FUNCTION_BLOCK FB_Machine EXTENDS FB_PackML_BaseModule // IMPLEMENTS I_ControlsProductionRate
VAR
    // Sub Modules
    GantryXYZ   : FB_GantryXYZ  := (Name := 'Gantry', LogStateChanges := TRUE);

    //Initial List of Components
    ipComponents_Init : ARRAY[1..Parameters_PackML_Base.MAX_NO_OF_COMPONENTS] OF I_ComponentBase := [];

	//Alarms for this module
	MachineAlarms : ARRAY[1..MACHINE_ALARM_COUNT] OF FB_TcAlarm;

END_VAR

VAR CONSTANT
    MACHINE_ALARM_COUNT : INT := 6;
END_VAR


METHOD PROTECTED Clearing
VAR
	i				: UDINT;
	SubModulesReady : BOOL := TRUE;
END_VAR
CASE SequenceState OF
    0:
        NoStateTasksToComplete := FALSE;
        SequenceState          := SequenceState + 10;
    10:
		//Leave Aborted thanks to this
		MachineAlarms[E_Seedra.EmergencyStop].Clear(0, 0);
        SequenceState := SequenceState + 10;
    20:

		SequenceState := SequenceState + 10;
	30: 
	
		SequenceState := SequenceState + 10;
	40:
		StateTasksComplete := TRUE; 
			 
END_CASE

SUPER^.Clearing();
END_METHOD

METHOD PROTECTED CreateEvents
VAR_INPUT
END_VAR
// Add your event creation here
F_CreateAllEventsInClass(Alarms     := MachineAlarms,
                         ClassSize  := SIZEOF(TC_Events.Seedra),
                         pInitEvent := ADR(TC_EVENTS.Seedra.InitReferenceEvent),
                         Prefix     := Name);
// Super call to base
SUPER^.CreateEvents();
END_METHOD

METHOD CyclicLogic
VAR_INPUT
END_VAR

IF NOT _InitComplete THEN
    _InitComplete := Initialize();
    RETURN;
END_IF

SUPER^.CyclicLogic();

//Here the alarms will raise and clear on its own if the input changes

//NOT GVL_Safety.eStopButton -> We Decouple physical button to Activate
  
IF GVL_Safety.eStopHMI OR NOT GVL_Safety.eStopButton AND NOT MachineAlarms[E_Seedra.EmergencyStop].bRaised THEN
	THIS^.ChangeState(E_PMLCommand.ePMLCommand_Abort);
	RaiseAlarmWithStrings(MachineAlarms[E_Seedra.EmergencyStop],'','');
//	ELSIF NOT GVL_Safety.eStop THEN
//	MachineAlarms[E_Seedra.EmergencyStop].Clear(0, 0);

END_IF
END_METHOD

METHOD PROTECTED Execute
CASE _CurrentMode OF

	//=================================PRODUCTION MODE==================================
	E_PMLUnitMode.ePMLUnitMode_Production:
		CASE SequenceState OF
			0:
				NoStateTasksToComplete := FALSE;

				//Advance Gantry to Resetting (Homing)
				GantryXYZ.ChangeState(E_PMLCommand.ePMLCommand_Start);
				
				SequenceState := SequenceState + 10;
					
			10:
				StateTasksComplete := TRUE;
				StateComplete();
				
			
		END_CASE

	//=================================MAINTENANCE & MANUAL MODE==================================
	E_PMLUnitMode.ePMLUnitMode_Maintenance, E_PMLUnitMode.ePMLUnitMode_Manual:
		;
END_CASE
END_METHOD

//! @summary Provides interlocks for HMI control and updates HMI status information for this module
METHOD PROTECTED HMICommunication

//! @description This method is called cyclically by <c>CyclicLogic()</c>

IF GVL_Safety.eStopHMI THEN
	PackMLBaseModule_HMI.Status.Error := TRUE;
	THIS^._Error := TRUE;
END_IF



SUPER^.HMICommunication();
END_METHOD

METHOD PROTECTED HMIPermissions
//General Mode Based Monitoring and handling of HMI control
CASE _CurrentMode OF
   
 E_PMLUnitMode.ePMLUnitMode_Production:
        CASE _CurrentState OF
            E_PMLState.ePMLState_Stopped:
				AllowHMIControl(ThisModuleOnly := FALSE);
            E_PMLState.ePMLState_Idle:
				AllowHMIControl(ThisModuleOnly := FALSE);
            E_PMLState.ePMLState_Suspended:
         		AllowHMIControl(ThisModuleOnly := FALSE);
            E_PMLState.ePMLState_Execute:
            	AllowHMIControl(ThisModuleOnly := FALSE); 
            E_PMLState.ePMLState_Aborted:
                AllowHMIControl(ThisModuleOnly := FALSE); 
            E_PMLState.ePMLState_Held:
                AllowHMIControl(ThisModuleOnly := FALSE); 
            E_PMLState.ePMLState_Complete:
          		AllowHMIControl(ThisModuleOnly := FALSE); 
        END_CASE
		
    E_PMLUnitMode.ePMLUnitMode_Manual:
        AllowHMIControl(ThisModuleOnly := FALSE); 
	E_PMLUnitMode.ePMLUnitMode_Maintenance:
        AllowHMIControl(ThisModuleOnly := FALSE); 
END_CASE
END_METHOD

METHOD PROTECTED Initialize : BOOL
VAR
    i : UDINT; //Generic iteration value
END_VAR
Initialize := FALSE;
CASE DescendantSequenceState OF
    0:
		RegisterSubmodule(GantryXYZ);

        _LogModeChanges         := FALSE;
        _LogStateChanges        := FALSE;
  
	    DescendantSequenceState := DescendantSequenceState + 10;
    10:
        DescendantSequenceState := DescendantSequenceState + 10;
    20:
        //Copy Mode names
        FOR i := 1 TO 3 DO
            ModeNames[i] := F_UnitModeToString(UDINT_TO_DINT(i));
        END_FOR

        DescendantSequenceState := DescendantSequenceState + 10;
    30:
        // Initialize Safety
		IF NOT GVL_Safety.RunStop THEN
			GVL_Safety.RunStop := TRUE;	
		END_IF
        DescendantSequenceState := DescendantSequenceState + 10;
    40:
        //Call the Super
        IF SUPER^.Initialize() THEN
            DescendantSequenceState := DescendantSequenceState + 10;
        END_IF

    50:
        Initialize := TRUE;
END_CASE
END_METHOD

METHOD PROTECTED Resetting
VAR
	i				: UDINT;
	SubModulesReady : BOOL := TRUE;
END_VAR
CASE _CurrentMode OF

	//=================================PRODUCTION MODE==================================
	E_PMLUnitMode.ePMLUnitMode_Production:
		CASE SequenceState OF
			0:
				NoStateTasksToComplete := FALSE;

				//Advance Gantry to Resetting (Homing)
				GantryXYZ.ChangeState(E_PMLCommand.ePMLCommand_Reset);
				
				SequenceState := SequenceState + 10;
					
			10:
				StateTasksComplete := TRUE;
				SUPER^.Resetting();
				
			
		END_CASE

	//=================================MAINTENANCE & MANUAL MODE==================================
	E_PMLUnitMode.ePMLUnitMode_Maintenance, E_PMLUnitMode.ePMLUnitMode_Manual:
		;
END_CASE
END_METHOD

//! @summary This method monitors <b>submodules</b> within this PackML module and initiates fault responses as required
METHOD PROTECTED SubModuleMonitor : BOOL
VAR
	AlarmResponses : ARRAY[0..4] OF E_AlarmResponse; //Temporary response array	
	i			   : UDINT;
END_VAR

//! @description This method is called cyclically by <c>CyclicLogic()</c>
// Check the sub Modules for Alarm Severity
SUPER^.SubModuleMonitor();

//Check the alarms at the machine level
_CurrentAlarmSeverity := F_GetMaxSeverityRaised(Alarms := MachineAlarms, CurrentSeverity := _CurrentAlarmSeverity);

//Check the severity of the machine level alarms
IF _CurrentState <> E_PMLState.ePMLState_Aborted AND _CurrentState <> E_PMLState.ePMLState_Aborting AND _CurrentState <> E_PMLState.ePMLState_Clearing  AND
   _CurrentState <> E_PMLState.ePMLState_Stopped AND _CurrentState <> E_PMLState.ePMLState_Stopping THEN
    AlarmResponses := _ParentFaultResponseDefinitions;
    CASE AlarmResponses[CurrentAlarmSeverity] OF
        E_AlarmResponse.Abort_ImmediateError:
            AbortImmediateError(Name, TRUE);
			AbortImmediateError(Name, FALSE);
        E_AlarmResponse.Abort_Immediate:
            AbortImmediate();
        E_AlarmResponse.Stop_Immediate:
            StopImmediate();
        E_AlarmResponse.Stop_Controlled:
            StopControlled();
        E_AlarmResponse.Hold_Immediate:
            HoldImmediate();
        E_AlarmResponse.Suspend_Immediate:
            SuspendImmediate();
        E_AlarmResponse.Suspend_Controlled:
            SuspendControlled();
        E_AlarmResponse.NoResponse:
            ;
    END_CASE
ELSIF _CurrentState = E_PMLState.ePMLState_Stopped OR _CurrentState = E_PMLState.ePMLState_Stopping THEN
    AlarmResponses := _ParentFaultResponseDefinitions;
    CASE AlarmResponses[CurrentAlarmSeverity] OF
        E_AlarmResponse.Abort_ImmediateError:
            AbortImmediateError(Name, TRUE);
        E_AlarmResponse.Abort_Immediate:
            AbortImmediate();
        E_AlarmResponse.NoResponse:
            ;
    END_CASE
END_IF
END_METHOD

END_FUNCTION_BLOCK

(* stored: Version 1.1.0.1, ProductVersion 3.1.4024.15
   POU FB_Machine: Id {dbe4ab41-c30f-0405-3dd0-3ec2a0f1563b}, SpecialFunc None
   Folder States: Id {70644f5e-d79a-440d-8d18-4948c059f975}
   Method Clearing: Id {309e3014-c1be-40c6-8306-4211d554a87f}
   Method CreateEvents: Id {30d2271a-6055-0dca-0156-9f862888fbc8}
   Method CyclicLogic: Id {340a2930-ae35-0e59-083f-71f30be69564}
   Method Execute: Id {729254ca-03f3-4bb9-98a5-84b797a61e6c}
   Method HMICommunication: Id {1b236574-a3d3-4f3d-8766-b10300116b01}
   Method HMIPermissions: Id {0fd4a0c7-5439-0f75-270c-fc092be30ec0}
   Method Initialize: Id {c6c0b1d2-c664-0498-029b-8500b66bc9b3}
   Method Resetting: Id {e510dc83-237a-4a59-97e9-db4b9408b4b7}
   Method SubModuleMonitor: Id {05824ff8-f244-497a-8a5d-923cd9a5fc87} *)
